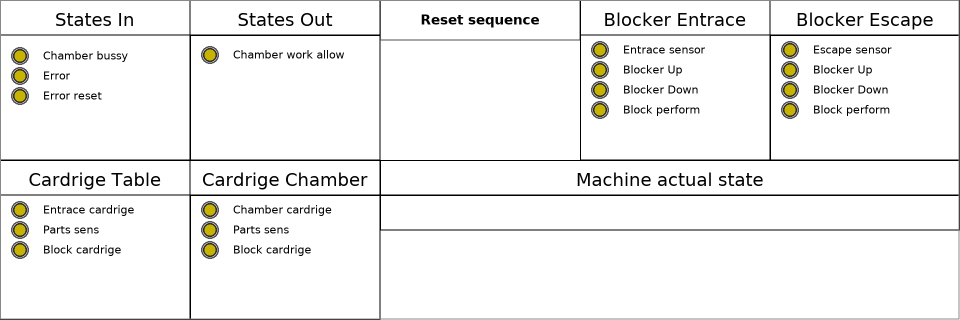
VISUALIZATION vTransporterFrame_V2  // 960x320
VAR_IN_OUT
	stData 		: stTransporterInOuts;
	stStatus	: stUnderPressureTestStatus_V2;
	iWorkStep	: INT;
END_VAR
    Rectangle (190,35 190x125)
    Rectangle (0,0 190x160)
    Rectangle (580,0 380x35)
    Lamp1 (10,46 20x20), variable: stStatus.bBusy, style: Lamp-Lamp1-Yellow
    Lamp1 (10,66 20x20), variable: stStatus.bError, style: Lamp-Lamp1-Yellow
    Lamp1 (10,86 20x20), variable: NOT stStatus.bError, style: Lamp-Lamp1-Yellow
    Label (40,46 150x20), "Chamber bussy"
    Label (40,66 150x20), "Error"
    Label (40,86 150x20), "Error reset"
    Lamp1 (200,45 20x20), variable: stStatus.bWorkAllow, style: Lamp-Lamp1-Yellow
    Label (230,45 150x20), "Chamber work allow"
    Rectangle (0,0 380x35)
    Label (0,5 190x30), "States In"
    Label (190,5 190x30), "States Out"
    Rectangle (380,0 200x40), "Reset sequence", input disabled if: NOT GVL.fbUserLogin.bPermissionGranted
        OnMouseClick: execute { stStatus.bResetSequence := TRUE; }
    Label (770,5 190x30), "Blocker Escape"
    Rectangle (580,0 190x160)
    Rectangle (770,35 190x125)
    Label (580,5 190x30), "Blocker Entrace"
    Rectangle (0,160 380x35)
    Label (190,165 190x30), "Cardrige Chamber"
    Rectangle (0,160 190x160)
    Rectangle (190,195 190x125)
    Label (0,165 190x30), "Cardrige Table"
    Label (620,40 150x20), "Entrace sensor"
    Lamp1 (590,40 20x20), variable: stData.bEntraceCarriage, style: Lamp-Lamp1-Yellow
    Lamp1 (590,60 20x20), variable: stData.bBlockerEntryUp, style: Lamp-Lamp1-Yellow
    Lamp1 (590,80 20x20), variable: stData.bBlockerEntryDown, style: Lamp-Lamp1-Yellow
    Lamp1 (590,100 20x20), variable: stData.bEntraceBlocker, style: Lamp-Lamp1-Yellow
    Label (620,60 150x20), "Blocker Up"
    Label (620,80 150x20), "Blocker Down"
    Label (620,100 150x20), "Block perform"
    Label (810,40 150x20), "Escape sensor"
    Lamp1 (780,40 20x20), variable: stData.bEscapeSensor, style: Lamp-Lamp1-Yellow
    Lamp1 (780,60 20x20), variable: stData.bBlockerEscapeUp, style: Lamp-Lamp1-Yellow
    Lamp1 (780,80 20x20), variable: stData.bBlockerEscapeDown, style: Lamp-Lamp1-Yellow
    Lamp1 (780,100 20x20), variable: stData.bEscapeBlocker, style: Lamp-Lamp1-Yellow
    Label (810,60 150x20), "Blocker Up"
    Label (810,80 150x20), "Blocker Down"
    Label (810,100 150x20), "Block perform"
    Label (40,200 150x20), "Entrace cardrige"
    Lamp1 (10,200 20x20), variable: stData.bEntraceCarriage, style: Lamp-Lamp1-Yellow
    Lamp1 (10,220 20x20), variable: stData.bPartsEntraceCarriage, style: Lamp-Lamp1-Yellow
    Lamp1 (10,240 20x20), variable: stData.bCarriageBlockerEntrace, style: Lamp-Lamp1-Yellow
    Label (40,220 150x20), "Parts sens"
    Label (40,240 150x20), "Block cardrige"
    Label (230,200 150x20), "Chamber cardrige"
    Lamp1 (200,200 20x20), variable: stData.bEntraceChamber, style: Lamp-Lamp1-Yellow
    Lamp1 (200,220 20x20), variable: stData.bPartsEntraceChamber, style: Lamp-Lamp1-Yellow
    Lamp1 (200,240 20x20), variable: stData.bCarriageBlockerChamber, style: Lamp-Lamp1-Yellow
    Label (230,220 150x20), "Parts sens"
    Label (230,240 150x20), "Block cardrige"
    Label (380,165 580x30), "Machine actual state"
    Rectangle (380,160 580x35)
    Rectangle (380,195 580x35), text list: 'tlTransporterSequence_V2', text index: iWorkStep
END_VISUALIZATION

(* stored: Version 1.1.0.1, ProductVersion 3.1.4024.13
   Visu vTransporterFrame_V2: Id {dbe8123b-8405-46ae-b721-ecfdb7d9fa20} *)
